// Mitsubishi GX Works2 project: PLC_26_Group_NEW   PLC: FX3G

// global labels: Global1
VAR_GLOBAL
  start_day_button AT X007 : BOOL;
  raspberry_input AT D1100 : REAL;
  raspberry_quantity AT D1102 : REAL;
  update_quantity AT M380 : BOOL;
  lemon_input AT D1200 : REAL;
  lemon_quantity AT D1202 : REAL;
  Stabilizer_input AT D1300 : REAL;
  Stabilizer_quantity AT D1302 : REAL;
  Gummy_bears_input AT D1400 : REAL;
  Gummy_bears_quantity AT D1402 : REAL;
  end_day_indicator AT M0 : BOOL;
  WORK_DAY_ACTIVE AT Y007 : BOOL;
  start_process AT X001 : BOOL;
  gumigum_type AT D1500 : REAL;
END_VAR
VAR_GLOBAL CONSTANT
  constant_400 : REAL := 400.0;
  div400 : REAL := 400.0;
END_VAR
VAR_GLOBAL
  maraz_type_check AT M10 : BOOL;
END_VAR
VAR_GLOBAL CONSTANT
  con_400 : REAL := 400.0;
END_VAR
VAR_GLOBAL
  AnalogInput1SIMULATION AT D2202 : INT;
END_VAR
VAR_GLOBAL CONSTANT
  con_5 : REAL := 5.0;
END_VAR
VAR_GLOBAL
  regular_maraz AT M4 : BOOL;
END_VAR
VAR_GLOBAL CONSTANT
  con_10 : REAL := 10.0;
  con_6 : REAL := 6.0;
END_VAR
VAR_GLOBAL
  pinuk_maraz AT M5 : BOOL;
END_VAR
VAR_GLOBAL CONSTANT
  con_280 : REAL := 280.0;
  con_455 : REAL := 455.0;
  con_105 : REAL := 105.0;
  con_28 : REAL := 28.0;
END_VAR
VAR_GLOBAL
  not_enough_for_regular AT M11 : BOOL;
END_VAR
VAR_GLOBAL CONSTANT
  con_385 : REAL := 385.0;
  con_665 : REAL := 665.0;
  con_210 : REAL := 210.0;
END_VAR
VAR_GLOBAL
  not_enough_for_pinuk AT M12 : BOOL;
  emergency_button AT X005 : BOOL;
  raspberry_container AT D1104 : REAL;
  lemon_container AT D1204 : REAL;
END_VAR
VAR_GLOBAL CONSTANT
  con_350 : REAL := 350.0;
  con_490 : REAL := 490.0;
  con_560 : REAL := 560.0;
  con_700 : REAL := 700.0;
END_VAR
VAR_GLOBAL
  TC AT TC0 : BOOL;
  TC_5_sec : BOOL;
END_VAR
VAR_GLOBAL CONSTANT
  con_50 : INT := 50;
END_VAR
VAR_GLOBAL
  TC0_5_sec AT TC0 : BOOL;
  TS_5sec AT TS0 : BOOL;
  ice_cream_in_progress AT Y000 : BOOL;
END_VAR
VAR_GLOBAL CONSTANT
  con_70 : REAL := 70.0;
END_VAR
VAR_GLOBAL
  start_cooling AT X002 : BOOL;
  raspberry_cooling_container AT D1106 : REAL;
  lemon_cooling_container AT D1206 : REAL;
  temperature_sensor AT X003 : BOOL;
  TC1_8_sec AT TC1 : BOOL;
END_VAR
VAR_GLOBAL CONSTANT
  con_80 : INT := 80;
END_VAR
VAR_GLOBAL
  TS_8sec AT TS1 : BOOL;
  ice_cream_in_cooling AT Y002 : BOOL;
END_VAR
VAR_GLOBAL CONSTANT
  con_0 : REAL;
END_VAR
VAR_GLOBAL
  finish_ice_cream_making AT M13 : BOOL;
  finish_cooling AT M14 : BOOL;
  mixing_container AT D2000 : REAL;
END_VAR
VAR_GLOBAL CONSTANT
  con_30 : INT := 30;
END_VAR
VAR_GLOBAL
  TC2_3sec AT TC2 : BOOL;
  TC3_5sec AT TC3 : BOOL;
  TS_3sec AT TS2 : BOOL;
  TS3_5sec AT TS3 : BOOL;
  blink_flag AT M15 : BOOL;
  TC4_1sec AT TC4 : BOOL;
END_VAR
VAR_GLOBAL CONSTANT
  con_10ms : INT := 10;
END_VAR
VAR_GLOBAL
  TS4_1sec AT TS4 : BOOL;
  blink1 AT Y005 : BOOL;
  TC5_1sec AT TC5 : BOOL;
  blink2 AT Y006 : BOOL;
  TS5_1sec AT TS5 : BOOL;
  finish_mixing AT M16 : BOOL;
  total_marazim AT D7000 : REAL;
END_VAR
VAR_GLOBAL CONSTANT
  con_1 : REAL := 1.0;
  con_40 : REAL := 40.0;
END_VAR
VAR_GLOBAL
  AnalogOutputSIMULATION AT D2204 : INT;
  AnalogInput1 AT D8280 : INT;
  AnalogOutput AT D8282 : INT;
  NISUY AT Y011 : BOOL;
END_VAR

// task Task_01 (event TRUE, interval 0, priority 31): POU_01

PROGRAM POU_01
(* structured ladder/FBD written out as ST: instructions are called as NAME(EN, inputs, outputs); _pN, _eN, _tN stand for wires *)
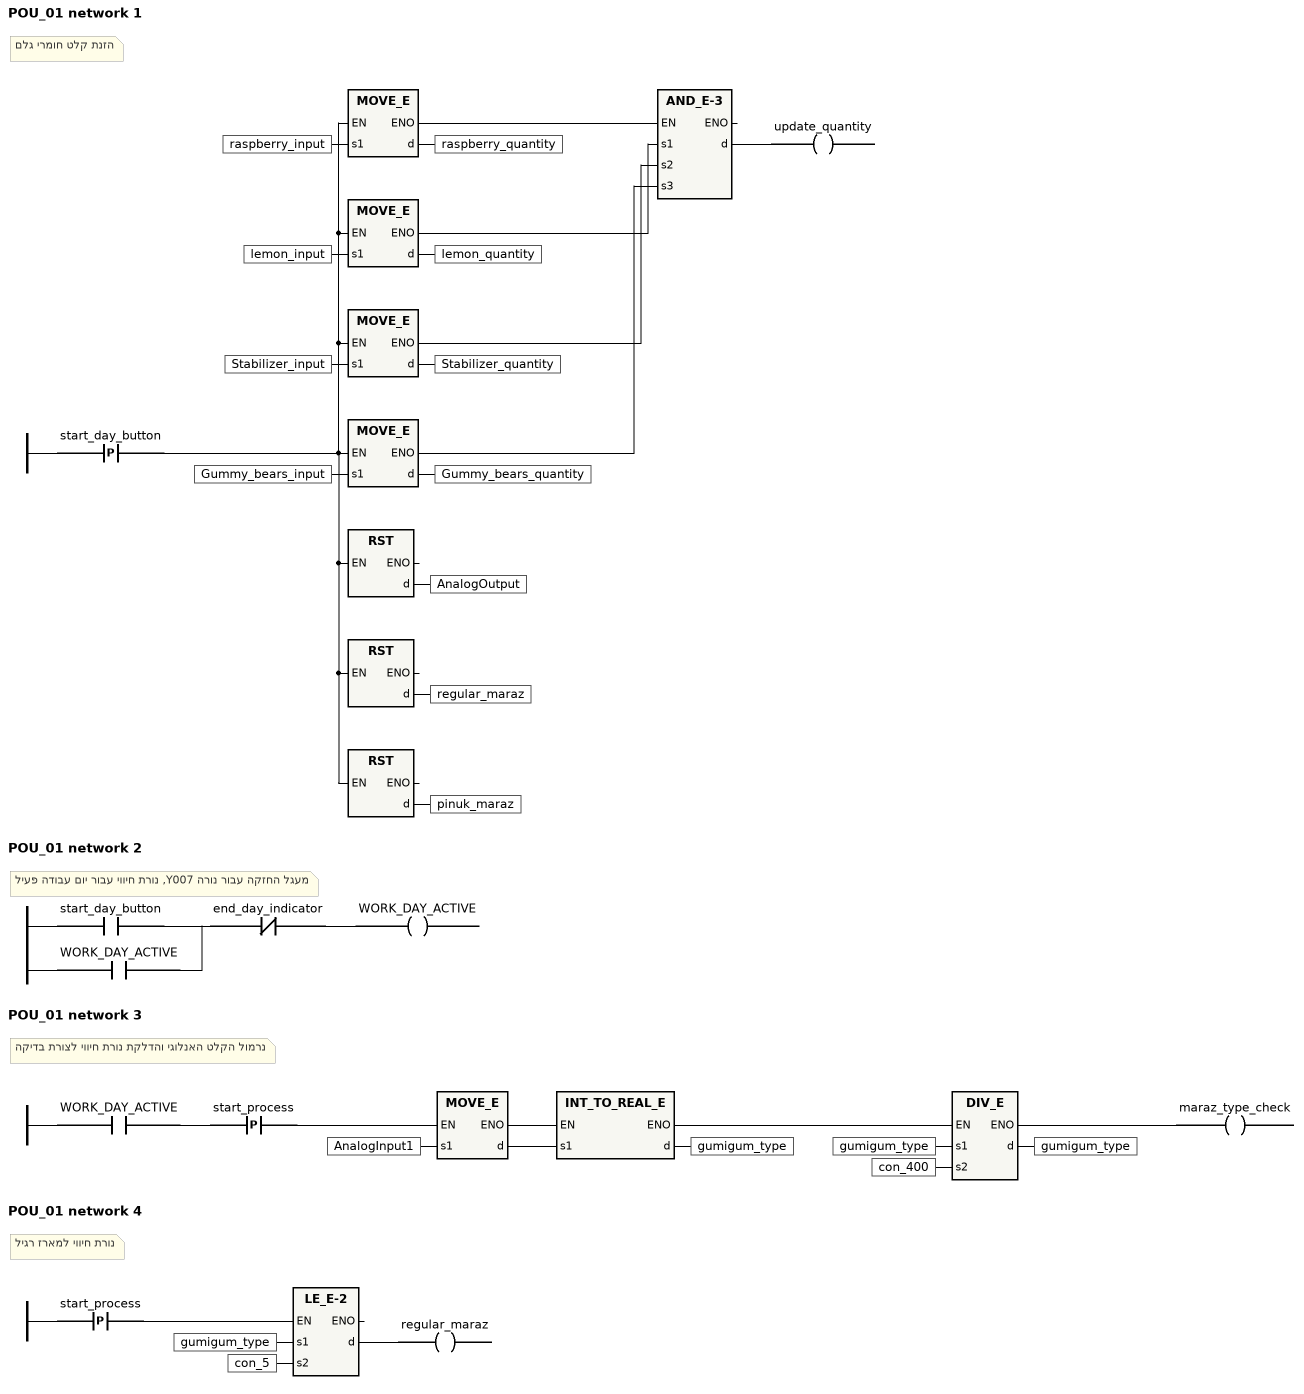
(* network 1 *)
(* הזנת קלט חומרי גלם *)
_p1 := LDP(TRUE, start_day_button);
_e2 := MOVE_E(_p1, raspberry_input, raspberry_quantity);
_e3 := MOVE_E(_p1, lemon_input, lemon_quantity);
_e4 := MOVE_E(_p1, Stabilizer_input, Stabilizer_quantity);
_e5 := MOVE_E(_p1, Gummy_bears_input, Gummy_bears_quantity);
AND_E(_e2, _e3, _e4, _e5, _t6);
update_quantity := _t6;
RST(_p1, AnalogOutput);
RST(_p1, regular_maraz);
RST(_p1, pinuk_maraz);
(* network 2 *)
(* מעגל החזקה עבור נורה Y007, נורת חיווי עבור יום עבודה פעיל *)
WORK_DAY_ACTIVE := (start_day_button OR WORK_DAY_ACTIVE) AND NOT end_day_indicator;
(* network 3 *)
(* נרמול הקלט האנלוגי והדלקת נורת חיווי לצורת בדיקה *)
_e2 := MOVE_E(WORK_DAY_ACTIVE AND LDP(TRUE, start_process), AnalogInput1, _t1);
_e3 := INT_TO_REAL_E(_e2, _t1, gumigum_type);
_e4 := DIV_E(_e3, gumigum_type, con_400, gumigum_type);
maraz_type_check := _e4;
(* network 4 *)
(* נורת חיווי למארז רגיל *)
LE_E(LDP(TRUE, start_process), gumigum_type, con_5, _t1);
regular_maraz := _t1;
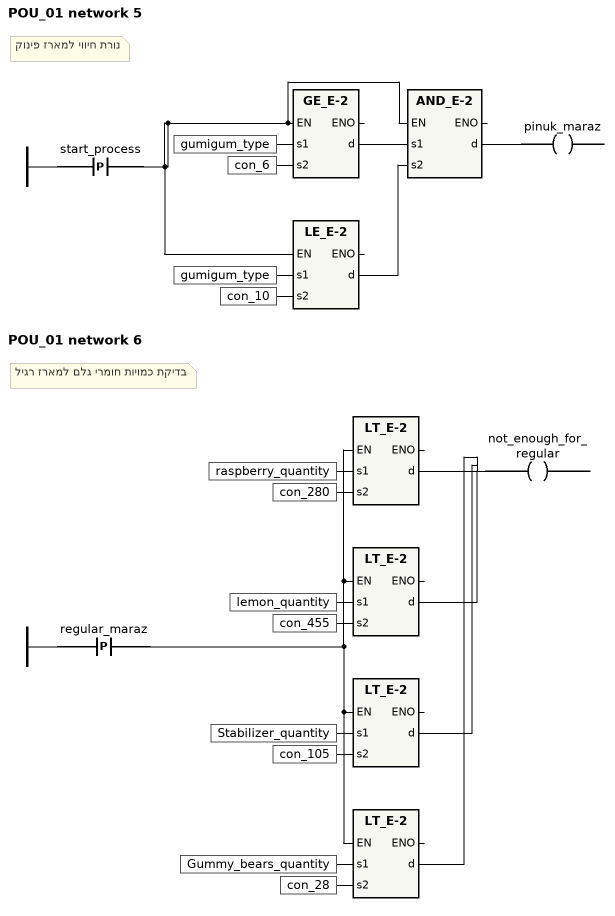
(* network 5 *)
(* נורת חיווי למארז פינוק *)
_p1 := LDP(TRUE, start_process);
GE_E(_p1, gumigum_type, con_6, _t2);
LE_E(_p1, gumigum_type, con_10, _t3);
AND_E(_p1, _t2, _t3, _t4);
pinuk_maraz := _t4;
(* network 6 *)
(* בדיקת כמויות חומרי גלם למארז רגיל *)
_p1 := LDP(TRUE, regular_maraz);
LT_E(_p1, raspberry_quantity, con_280, _t2);
LT_E(_p1, lemon_quantity, con_455, _t3);
LT_E(_p1, Stabilizer_quantity, con_105, _t4);
LT_E(_p1, Gummy_bears_quantity, con_28, _t5);
not_enough_for_regular := _t2 OR _t3 OR _t4 OR _t5;
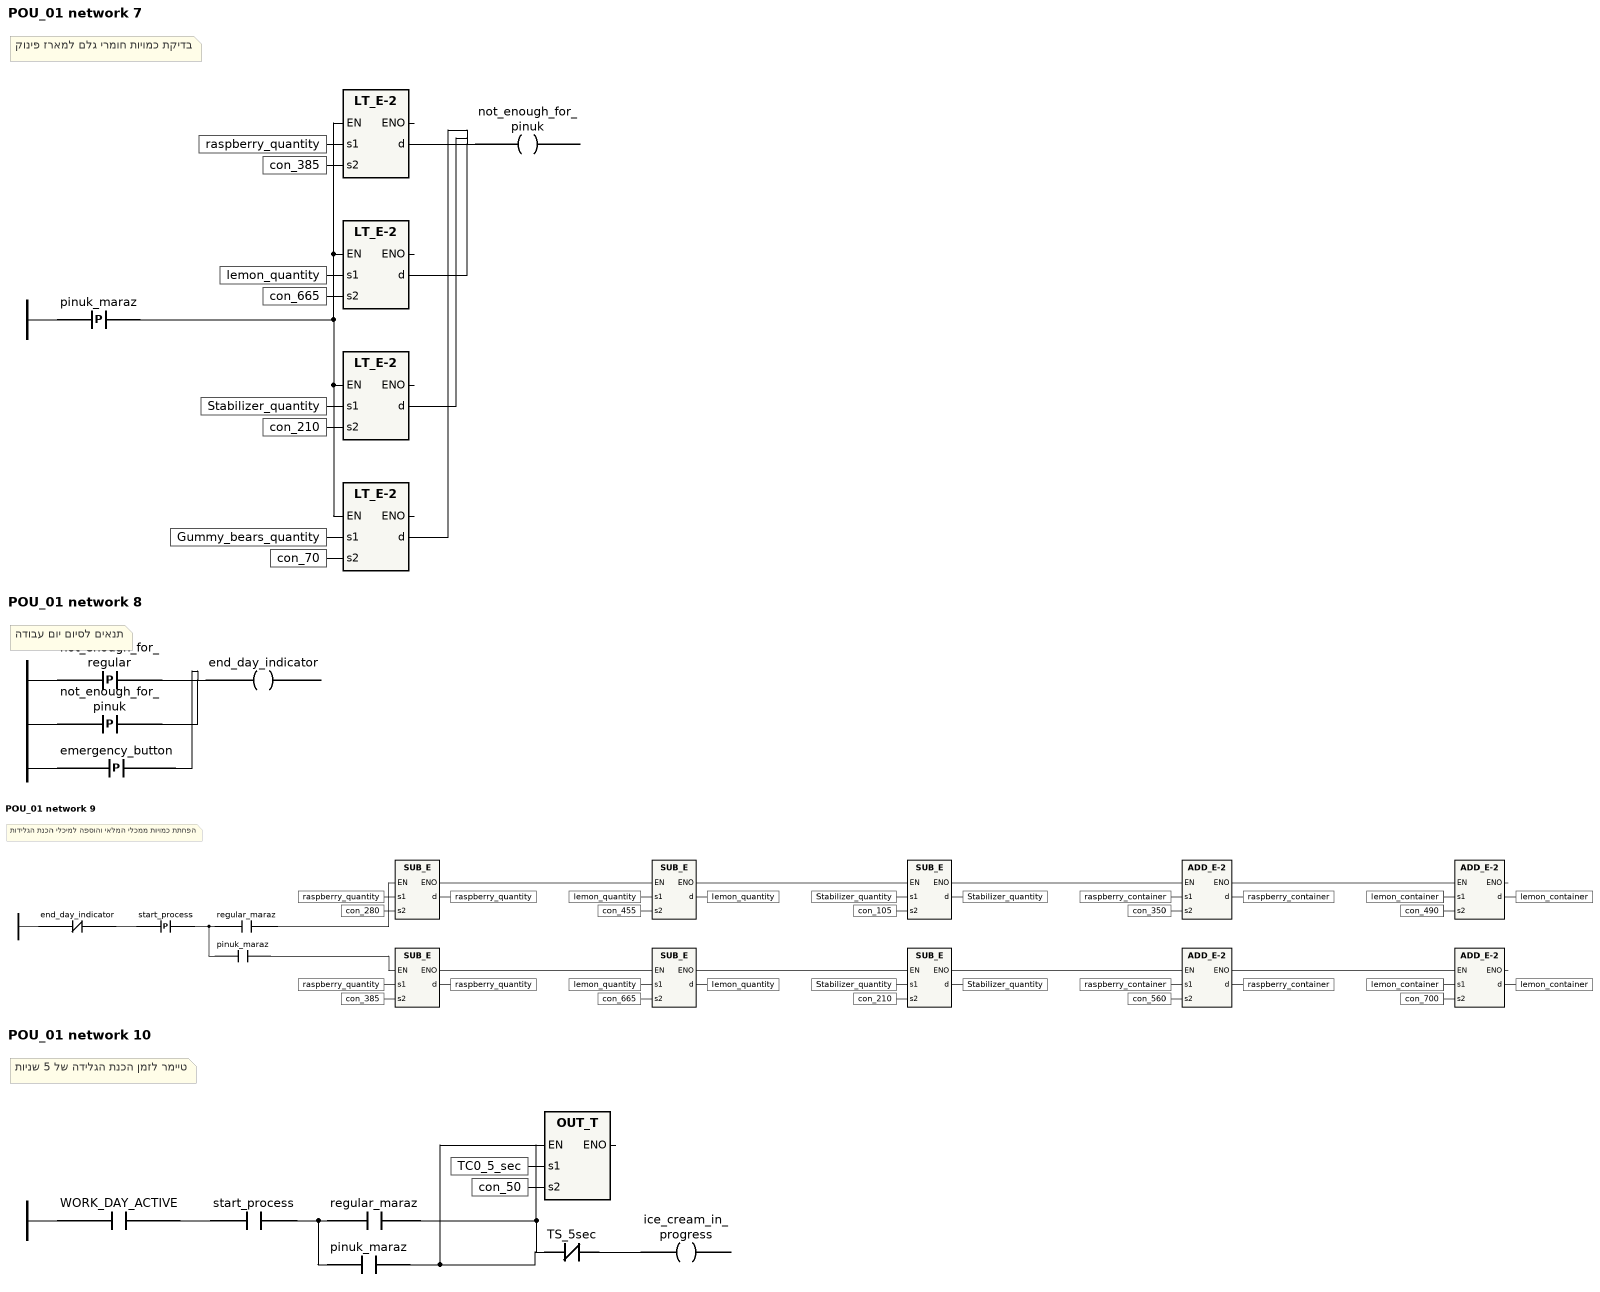
(* network 7 *)
(* בדיקת כמויות חומרי גלם למארז פינוק *)
_p1 := LDP(TRUE, pinuk_maraz);
LT_E(_p1, raspberry_quantity, con_385, _t2);
LT_E(_p1, lemon_quantity, con_665, _t3);
LT_E(_p1, Stabilizer_quantity, con_210, _t4);
LT_E(_p1, Gummy_bears_quantity, con_70, _t5);
not_enough_for_pinuk := _t2 OR _t3 OR _t4 OR _t5;
(* network 8 *)
(* תנאים לסיום יום עבודה *)
end_day_indicator := LDP(TRUE, not_enough_for_regular) OR LDP(TRUE, not_enough_for_pinuk) OR LDP(TRUE, emergency_button);
(* network 9 *)
(* הפחתת כמויות ממכלי המלאי והוספה למיכלי הכנת הגלידות *)
_p1 := NOT end_day_indicator AND LDP(TRUE, start_process);
_e2 := SUB_E(_p1 AND regular_maraz, raspberry_quantity, con_280, raspberry_quantity);
_e3 := SUB_E(_e2, lemon_quantity, con_455, lemon_quantity);
_e4 := SUB_E(_e3, Stabilizer_quantity, con_105, Stabilizer_quantity);
_e5 := ADD_E(_e4, raspberry_container, con_350, raspberry_container);
ADD_E(_e5, lemon_container, con_490, lemon_container);
_e6 := SUB_E(_p1 AND pinuk_maraz, raspberry_quantity, con_385, raspberry_quantity);
_e7 := SUB_E(_e6, lemon_quantity, con_665, lemon_quantity);
_e8 := SUB_E(_e7, Stabilizer_quantity, con_210, Stabilizer_quantity);
_e9 := ADD_E(_e8, raspberry_container, con_560, raspberry_container);
ADD_E(_e9, lemon_container, con_700, lemon_container);
(* network 10 *)
(* טיימר לזמן הכנת הגלידה של 5 שניות *)
_p1 := WORK_DAY_ACTIVE AND start_process;
_p2 := (_p1 AND regular_maraz) OR (_p1 AND pinuk_maraz);
OUT_T(_p2, TC0_5_sec, con_50);
ice_cream_in_progress := _p2 AND NOT TS_5sec;
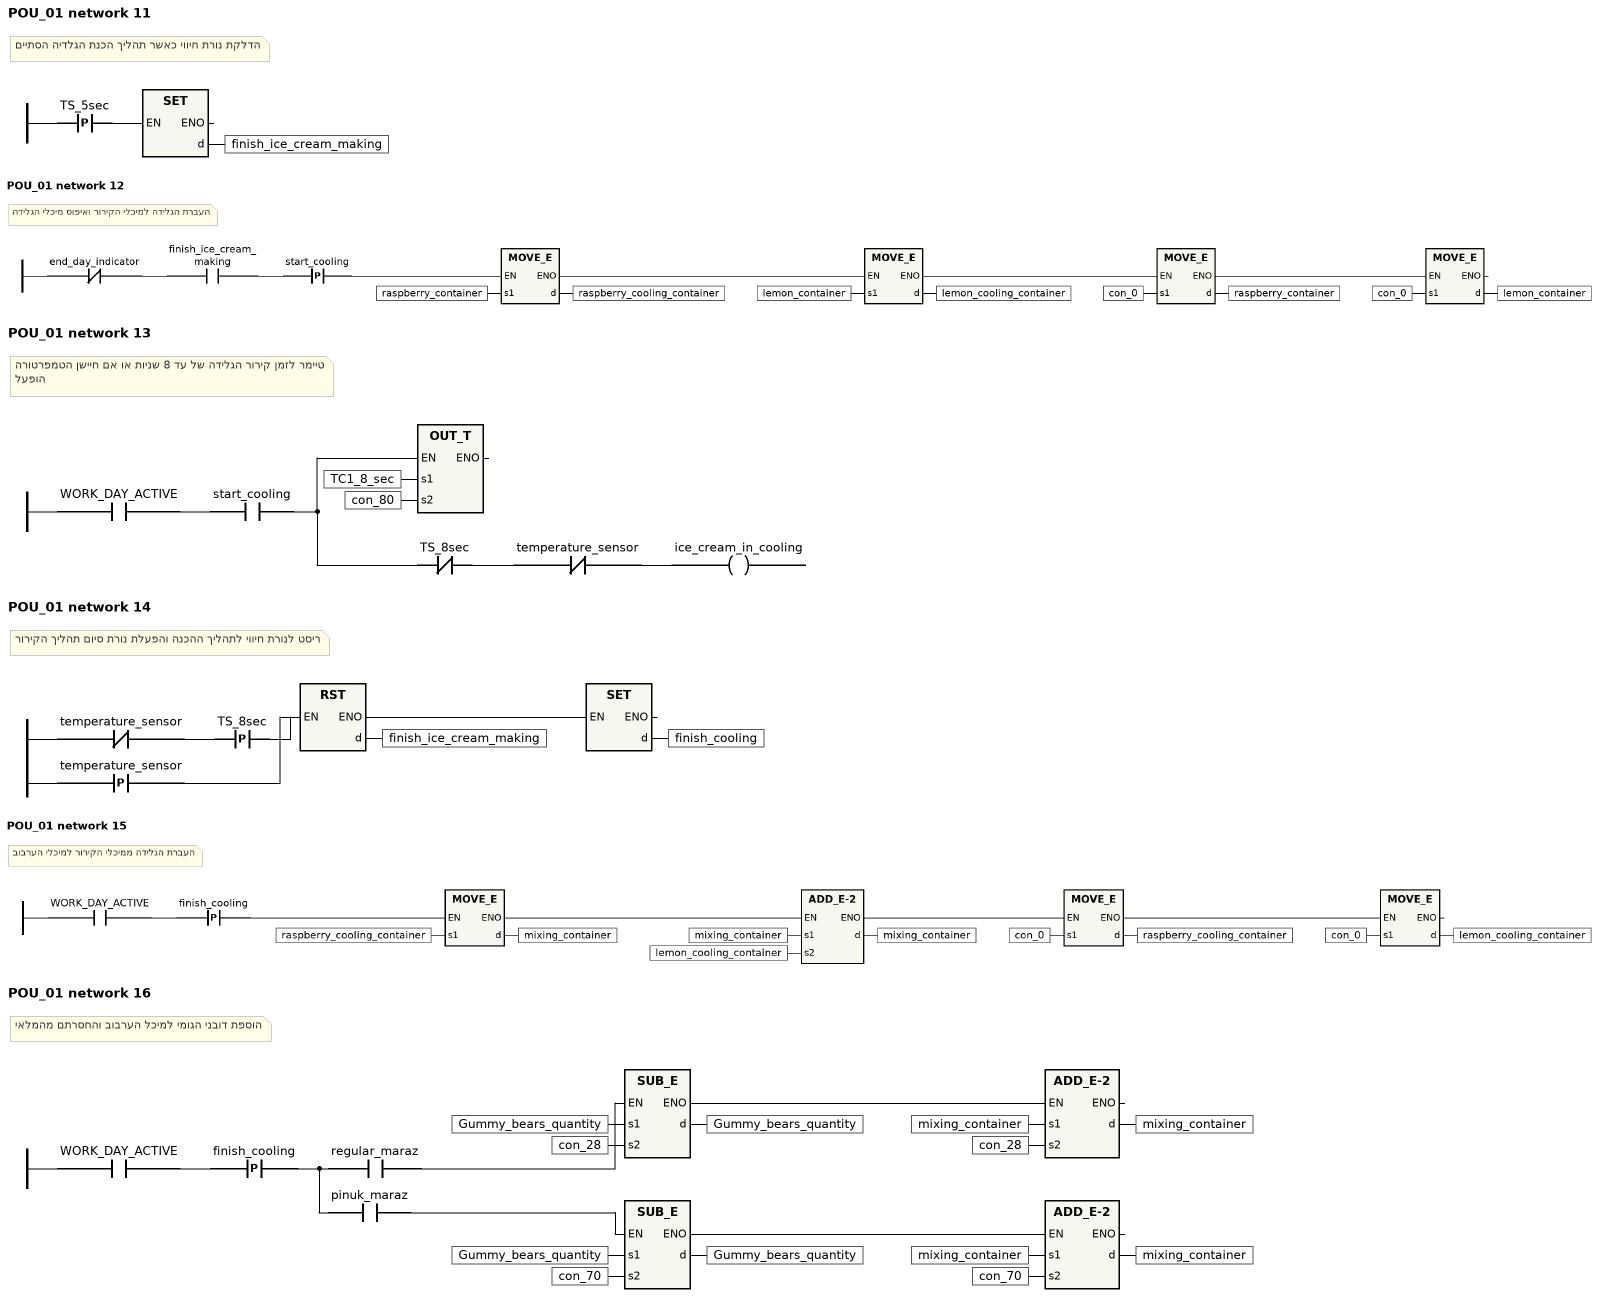
(* network 11 *)
(* הדלקת נורת חיווי כאשר תהליך הכנת הגלדיה הסתיים *)
SET(LDP(TRUE, TS_5sec), finish_ice_cream_making);
(* network 12 *)
(* העברת הגלידה למיכלי הקירור ואיפוס מיכלי הגלידה *)
_e1 := MOVE_E(NOT end_day_indicator AND finish_ice_cream_making AND LDP(TRUE, start_cooling), raspberry_container, raspberry_cooling_container);
_e2 := MOVE_E(_e1, lemon_container, lemon_cooling_container);
_e3 := MOVE_E(_e2, con_0, raspberry_container);
MOVE_E(_e3, con_0, lemon_container);
(* network 13 *)
(* טיימר לזמן קירור הגלידה של עד 8 שניות או אם חיישן הטמפרטורה הופעל *)
_p1 := WORK_DAY_ACTIVE AND start_cooling;
OUT_T(_p1, TC1_8_sec, con_80);
ice_cream_in_cooling := _p1 AND NOT TS_8sec AND NOT temperature_sensor;
(* network 14 *)
(* ריסט לנורת חיווי לתהליך ההכנה והפעלת נורת סיום תהליך הקירור *)
_e1 := RST((NOT temperature_sensor AND LDP(TRUE, TS_8sec)) OR LDP(TRUE, temperature_sensor), finish_ice_cream_making);
SET(_e1, finish_cooling);
(* network 15 *)
(* העברת הגלידה ממיכלי הקירור למיכלי הערבוב *)
_e1 := MOVE_E(WORK_DAY_ACTIVE AND LDP(TRUE, finish_cooling), raspberry_cooling_container, mixing_container);
_e2 := ADD_E(_e1, mixing_container, lemon_cooling_container, mixing_container);
_e3 := MOVE_E(_e2, con_0, raspberry_cooling_container);
MOVE_E(_e3, con_0, lemon_cooling_container);
(* network 16 *)
(* הוספת דובני הגומי למיכל הערבוב והחסרתם מהמלאי *)
_p1 := WORK_DAY_ACTIVE AND LDP(TRUE, finish_cooling);
_e2 := SUB_E(_p1 AND regular_maraz, Gummy_bears_quantity, con_28, Gummy_bears_quantity);
ADD_E(_e2, mixing_container, con_28, mixing_container);
_e3 := SUB_E(_p1 AND pinuk_maraz, Gummy_bears_quantity, con_70, Gummy_bears_quantity);
ADD_E(_e3, mixing_container, con_70, mixing_container);
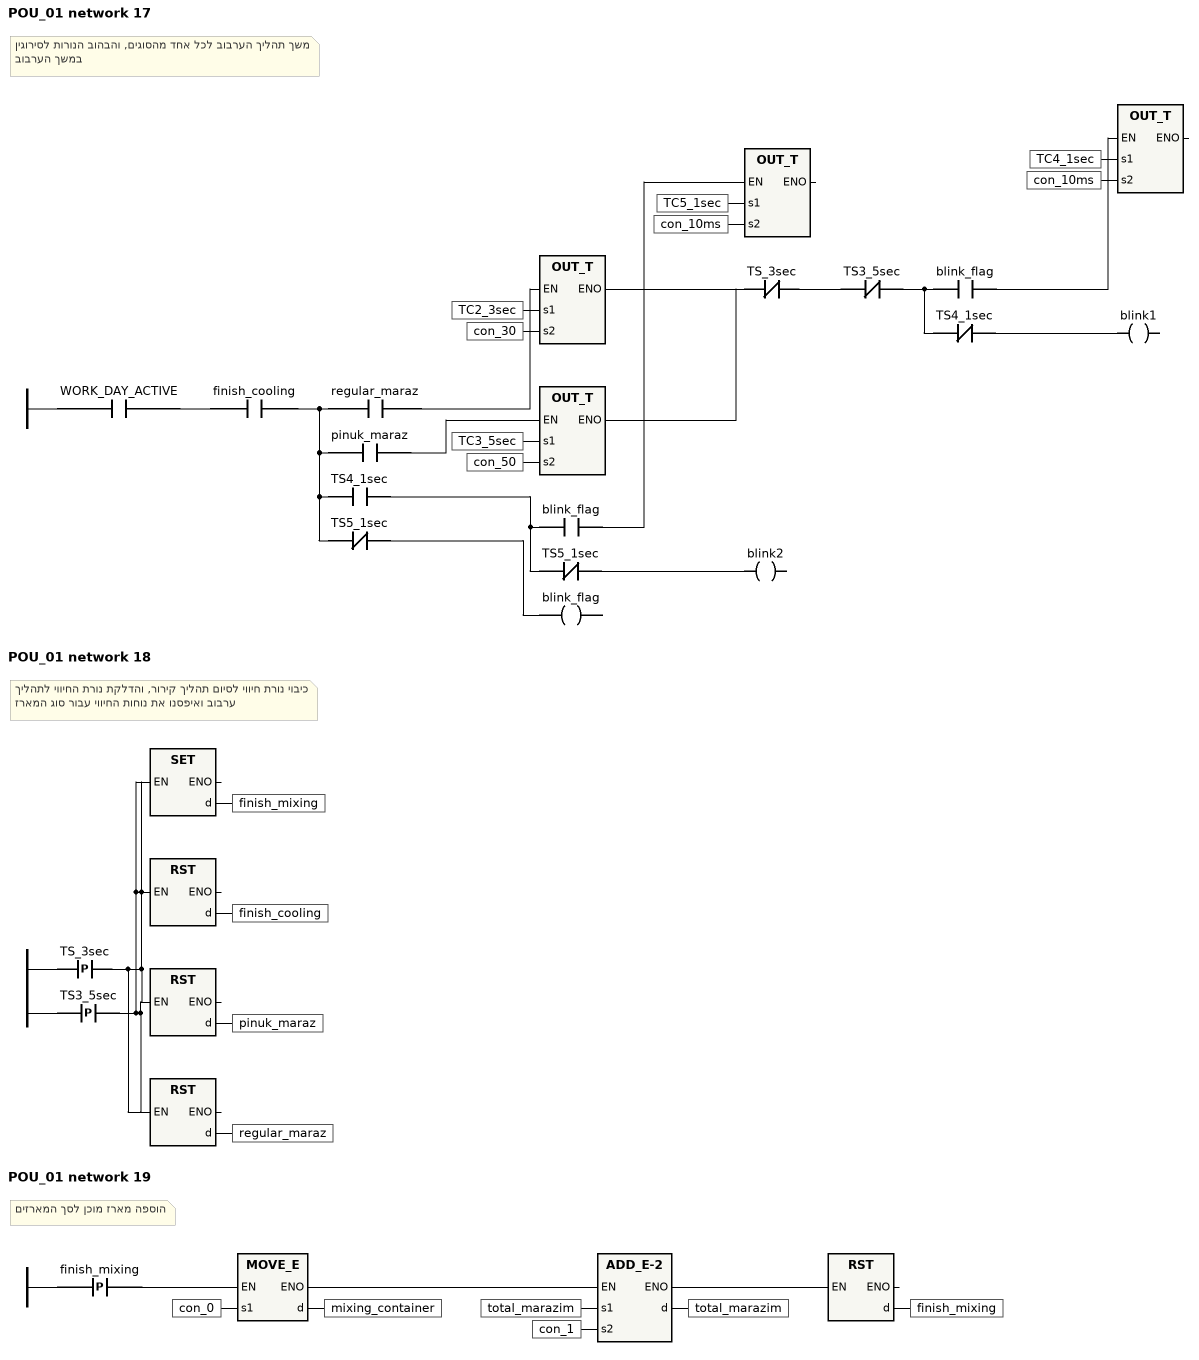
(* network 17 *)
(* משך תהליך הערבוב לכל אחד מהסוגים, והבהוב הנורות לסירוגין במשך הערבוב *)
_p1 := WORK_DAY_ACTIVE AND finish_cooling;
_e2 := OUT_T(_p1 AND regular_maraz, TC2_3sec, con_30);
_e3 := OUT_T(_p1 AND pinuk_maraz, TC3_5sec, con_50);
_p4 := ((_e2 OR _e3) AND NOT TS_3sec) AND NOT TS3_5sec;
OUT_T(_p4 AND blink_flag, TC4_1sec, con_10ms);
blink1 := _p4 AND NOT TS4_1sec;
_p5 := _p1 AND TS4_1sec;
OUT_T(_p5 AND blink_flag, TC5_1sec, con_10ms);
blink2 := _p5 AND NOT TS5_1sec;
blink_flag := _p1 AND NOT TS5_1sec;
(* network 18 *)
(* כיבוי נורת חיווי לסיום תהליך קירור, והדלקת נורת החיווי לתהליך ערבוב ואיפסנו את נוחות החיווי עבור סוג המארז *)
_p1 := LDP(TRUE, TS_3sec) OR LDP(TRUE, TS3_5sec);
SET(_p1, finish_mixing);
RST(_p1, finish_cooling);
RST(_p1, pinuk_maraz);
RST(_p1, regular_maraz);
(* network 19 *)
(* הוספה מארז מוכן לסך המארזים *)
_e1 := MOVE_E(LDP(TRUE, finish_mixing), con_0, mixing_container);
_e2 := ADD_E(_e1, total_marazim, con_1, total_marazim);
RST(_e2, finish_mixing);
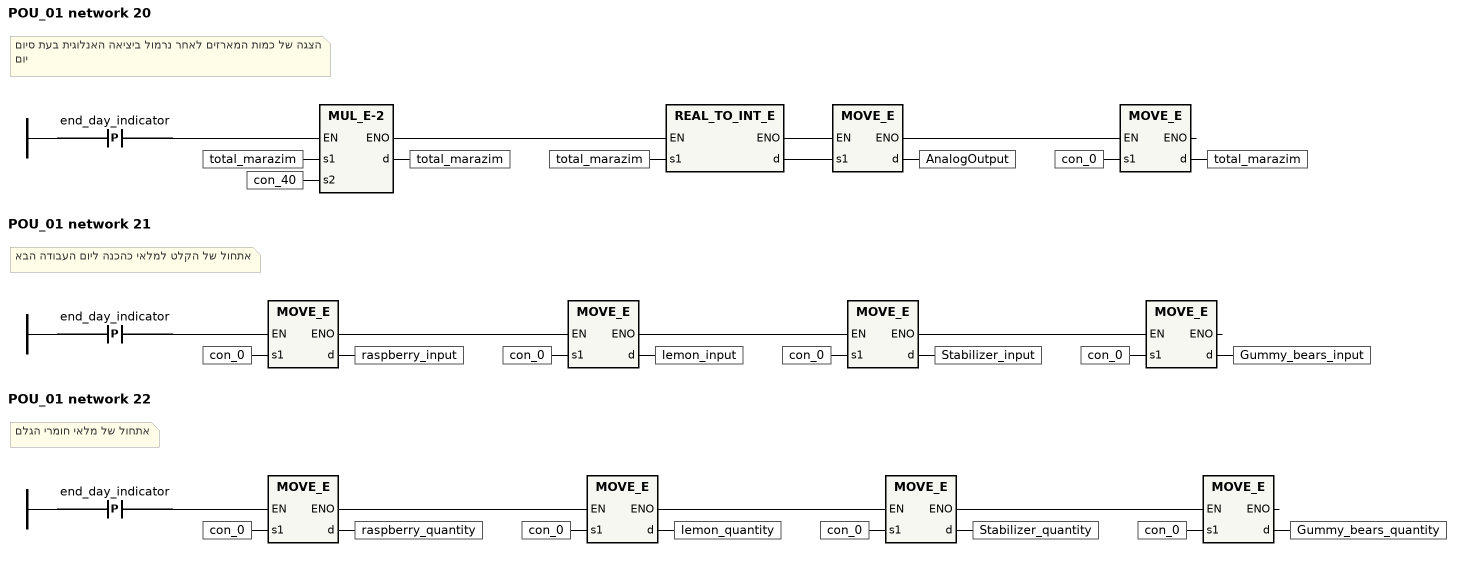
(* network 20 *)
(* הצגה של כמות המארזים לאחר נרמול ביציאה האנלוגית בעת סיום יום *)
_e1 := MUL_E(LDP(TRUE, end_day_indicator), total_marazim, con_40, total_marazim);
_e3 := REAL_TO_INT_E(_e1, total_marazim, _t2);
_e4 := MOVE_E(_e3, _t2, AnalogOutput);
MOVE_E(_e4, con_0, total_marazim);
(* network 21 *)
(* אתחול של הקלט למלאי כהכנה ליום העבודה הבא *)
_e1 := MOVE_E(LDP(TRUE, end_day_indicator), con_0, raspberry_input);
_e2 := MOVE_E(_e1, con_0, lemon_input);
_e3 := MOVE_E(_e2, con_0, Stabilizer_input);
MOVE_E(_e3, con_0, Gummy_bears_input);
(* network 22 *)
(* אתחול של מלאי חומרי הגלם *)
_e1 := MOVE_E(LDP(TRUE, end_day_indicator), con_0, raspberry_quantity);
_e2 := MOVE_E(_e1, con_0, lemon_quantity);
_e3 := MOVE_E(_e2, con_0, Stabilizer_quantity);
MOVE_E(_e3, con_0, Gummy_bears_quantity);
END_PROGRAM
